(*
SPDX-FileCopyrightText: © 2026 Oleksandr Tiutyk <trofimich@gmail.com>
SPDX-License-Identifier: MIT
License: https://opensource.org/license/mit
*)

(*!
<summary>Obtains the library namespace through the init_namespace attribute.</summary>
<description>
Internal static metadata holder. Its output is initialized by TwinCAT rather than by cyclic execution.
</description>
*)

FUNCTION_BLOCK INTERNAL NamespaceExtractor
VAR_OUTPUT
	{attribute 'init_namespace'} 
	CurrentNamespace : STRING;	
END_VAR

END_FUNCTION_BLOCK

(* stored: Version 1.1.0.1
   POU NamespaceExtractor: Id {ec23540e-4f6e-4415-bd00-943358bc77a2}, SpecialFunc None *)
